// TIA Portal V21 export
VAR_GLOBAL   // PLC tag table "K_Popups"
END_VAR
VAR_GLOBAL CONSTANT   // user constants
   K_Popup_ConfermareCuboRimosso : Int := 1;
   K_Popup_ConfermareCambioAttrezzatura : Int := 2;
END_VAR
